Universal Robots URScript: Test Teach Position.script

def Test_Teach_Position():
  global _hidden_verificationVariable=0
  set_tool_communication(False, 115200, 0, 1, 1.5, 3.5)
  set_tool_output_mode(0)
  set_tool_digital_output_mode(0, 1)
  set_tool_digital_output_mode(1, 1)
  set_tool_voltage(0)
  set_gravity([0.0, 0.0, 9.82])
  set_safety_mode_transition_hardness(1)
  set_tcp(p[0.0,0.0,0.019,0.0,0.0,0.0])
  set_standard_analog_input_domain(0, 1)
  set_standard_analog_input_domain(1, 1)
  set_tool_analog_input_domain(0, 1)
  set_tool_analog_input_domain(1, 1)
  set_analog_outputdomain(0, 0)
  set_analog_outputdomain(1, 0)
  set_input_actions_to_default()
  set_target_payload(0.310000, [0.000000, 0.000000, 0.009500], [0.000219, 0.000219, 0.000219, 0.000000, 0.000000, 0.000000])
  global Point_1=p[0.0,0.0,0.0,0.0,0.0,0.0]
  # begin: URCap Installation Node
  #   Source: MachineLogic for Universal Robots, 3.1.7, Vention Inc.
  #   Type: MachineLogic for Universal Robots
  def waitForResponse(expected_response_vention, cname_vention):
  response_vention = socket_read_string(cname_vention,timeout=15)
  while response_vention != expected_response_vention:
  sleep(0.01)
  response_vention = socket_read_string(cname_vention,timeout=15)
  end
  sleep(0.01)
  sync()
  end
  def sendString(string_vention, expected_response_vention, cname_vention):
  socket_send_string(str_cat(string_vention,";"), cname_vention)
  response_vention = socket_read_string(cname_vention,timeout=15)
  if(response_vention == "nAck"):
  popup("nAck received")
  end
  while response_vention != expected_response_vention:
  sleep(0.01)
  response_vention = socket_read_string(cname_vention,timeout=15)
  if(response_vention == "nAck"):
  popup("nAck received")
  end
  end
  sleep(0.01)
  sync()
  end
  def sendStringNAck(string_vention, expected_response_vention, cname_vention):
  socket_send_string(str_cat(string_vention,";"), cname_vention)
  response_vention = socket_read_string(cname_vention,timeout=15)
  if(response_vention == "nAck"):
  popup("nAck received")
  end
  while(response_vention != expected_response_vention and response_vention != "nAck"):
  sleep(0.01)
  response_vention = socket_read_string(cname_vention,timeout=15)
  if(response_vention == "nAck"):
  popup("nAck received",blocking=True)
  end
  end
  sleep(0.01)
  sync()
  end
  def sendStringWithTimeout(string_vention, expected_response_vention, cname_vention):
  socket_send_string(str_cat(string_vention,";"), cname_vention)
  response_vention = socket_read_string(cname_vention,timeout=10)
  if(response_vention == "nAck"):
  popup("nAck received"+string_vention)
  end
  sleep(0.01)
  sync()
  end
  def pollString(string_vention, expected_response_vention, cname_vention):
  socket_send_string(str_cat(string_vention,";"), cname_vention)
  response_vention = socket_read_string(cname_vention,timeout=15)
  if(response_vention == "nAck"):
  popup("nAck received")
  end
  while response_vention != expected_response_vention:
  sleep(1)
  socket_send_string(str_cat(string_vention,";"), cname_vention)
  response_vention = socket_read_string(cname_vention,timeout=15)
  if(response_vention == "nAck"):
  popup("nAck received")
  end
  end
  sleep(0.01)
  sync()
  end
  def sendVariable(var_vention, data_vention, expected_response_vention, cname_vention):
  socket_set_var(var_vention, data_vention, cname_vention)
  response_vention = socket_read_string(cname_vention,timeout=15)
  if(response_vention == "nAck"):
  popup("nAck received")
  end
  while response_vention != expected_response_vention:
  sleep(0.01)
  response_vention = socket_read_string(cname_vention,timeout=15)
  if(response_vention == "nAck"):
  popup("nAck received")
  end
  end
  sleep(0.01)
  sync()
  end
  def intToString(integer_vention,cname_vention):
  stringFix=""
  multiplier_vention123=1
  if integer_vention<0:
  stringFix="-"
  multiplier_vention123=-1
  end
  socket_set_var("GetString",integer_vention*multiplier_vention123,cname_vention)
  string_vention=""
  while string_vention=="":
  sleep(0.01)
  string_vention=socket_read_string(cname_vention,timeout=15)
  end
  sleep(0.01)
  sync()
  string_vention=stringFix+string_vention
  return string_vention
  end
  string_vention=""
  isVentionMovementBusy = False
  isVentionParallelMovementSendingScript = False
  ventionThreadHandle = 1
  isVentionMovementBusyMachineMotion1 = False
  isVentionParallelMovementSendingScriptMachineMotion1 = False
  socket_vention = socket_open("192.168.3.52", 9999, "MachineMotion1")
  if socket_vention==False:
  popup("Check configuration, can't connect to MachineMotion")
  end
  waitForResponse("MachineMotion connection established", "MachineMotion1")
  sendString("isReady", "MachineMotion isReady = true", "MachineMotion1")
  sendStringWithTimeout("setURCapVersion2", "setURCapVersion loaded", "MachineMotion1")
  sendString("SET speed_v2 1000000", "Ack", "MachineMotion1")
  sendString("SET acceleration_v2 100000", "Ack", "MachineMotion1")
  sendString("SET de_axis_1_microsteps_config 8", "Ack", "MachineMotion1")
  sendString("SET de_axis_1_mechanical_gain_config_v2 150000.0", "Ack", "MachineMotion1")
  sendString("SET de_axis_1_direction_config 1", "Ack", "MachineMotion1")
  sendString("SET de_axis_1_type_config Custom Actuator ", "Ack", "MachineMotion1")
  sendString("de_axis_1_config_exec", "Ack", "MachineMotion1")
  # end: URCap Installation Node
  step_count_25c65f44_06b5_40e8_ab7a_4740e82bbebb = 0.0
  thread Step_Counter_Thread_70793aa9_04f0_4a00_a81a_f8e9561ae1e6():
    while (True):
      step_count_25c65f44_06b5_40e8_ab7a_4740e82bbebb = step_count_25c65f44_06b5_40e8_ab7a_4740e82bbebb + 1.0
      sync()
    end
  end
  run Step_Counter_Thread_70793aa9_04f0_4a00_a81a_f8e9561ae1e6()
  global freedrive_m_var=  False
  global Waypoint_2_p=p[-.545552386461, .384638463642, .171639485768, .668511604681, -1.949272130073, 1.726627182696]
  global Waypoint_2_q=[-1.0565226713763636, -1.0868892234614869, 2.1878750959979456, -1.2335426074317475, -1.0471814314471644, 2.53226637840271]
  $ 13 "Thread_1"
  thread Thread_1():
    while (True):
      $ 14 "Loop  True "
      while (  True  ):
        $ 15 "If freedrive_m_var≟ True "
        if (freedrive_m_var ==   True  ):
          $ 16 "freedrive_mode()"
          freedrive_mode()
        else:
          $ 17 "Else" "noBreak"
          $ 18 "end_freedrive_mode()"
          end_freedrive_mode()
        end
        $ 19 "sync()"
        sync()
      end
    end
  end
  threadId_Thread_1 = run Thread_1()
  $ 2 "Robot Program"
  $ 3 "Home"
  movej([-2.5278157671606145, -1.852465766610969, 2.7650339410037645, -2.482569784177298, -1.5711424260709022, 2.183095047178716], a=1.3962634015954636, v=1.0471975511965976)
  $ 4 "MoveJ"
  $ 5 "Waypoint_2" "breakAfter"
  movej(get_inverse_kin(Waypoint_2_p, qnear=Waypoint_2_q), a=1.3962634015954636, v=1.0471975511965976)
  $ 6 "freedrive_m_var≔ False "
  global freedrive_m_var=  False
  $ 7 "freedrive_m_var≔ True "
  global freedrive_m_var=  True
  $ 8 "Popup: Move the robot to the peg center, then click 'Continue'"
  popup("Move the robot to the peg center, then click 'Continue'", "Message", False, False, blocking=True)
  $ 9 "freedrive_m_var≔ False "
  global freedrive_m_var=  False
  $ 10 "Wait: 0.25"
  sleep(0.25)
  $ 11 "sync()"
  sync()
  $ 12 "tcp_pose≔get_actual_joint_positions()"
  global tcp_pose= get_actual_joint_positions ()
end
